(*********************************** G.D S.p.A. - Technical Department ***********************************
============= PROGRAM INFO ============
FOLDER:             TBD
MACHINES INVOLVED:  TBD 

============= DESCRIPTION =============
csp machine declaration

============= REVISIONS ===============
Date		Version	 	Author      	Description             
----------	-------		------------  	--------------------------------------------
2019/04/05 	0000.00	 	M.Grasso		Creation of the PRG

**********************************************************************************************************)
(*$R process_ref := prc; $*)
PROGRAM csp_case_transport_ls
VAR
	
	prc:											process;
	prc_path:										STRING;
	
END_VAR

_read_var_input();

_object_manager();

IF NOT objects_running()
THEN
	RETURN;	
END_IF

_read_process_image();

_mode_manager();

_set_runtime_properties();

(********************************* BODY *********************************)
(************************************************************************)

_handle_messages();

_write_output();

ACTION _handle_messages:
;
END_ACTION

ACTION _handle_process_test:
;
END_ACTION

ACTION _mode_manager:
IF process_mode_req_is_pending(prc)
THEN
    process_apply_mode_req_first_step(prc);
    CASE process_get_mode(prc) OF
        MODE_TO_ABSENT:
			;
        MODE_TO_INACTIVE:
			;
        MODE_TO_TEST:
			;
        MODE_TO_OPERATIONAL:
			;
    END_CASE
    process_apply_mode_req_second_step(prc);
END_IF
END_ACTION

ACTION _object_manager:
IF objects_initialization()
THEN
	sub_process_init(
		object_name					:= 'csp_case_transport_ls.prc', 
		process						:= csp_case_transport.prc, 
		CONVERSION_this				:= prc);
		
	prc_path 						:= process_get_path(prc);
END_IF

IF objects_running()
THEN
	process_cycle(prc);
END_IF
END_ACTION

ACTION _read_process_image:
;
END_ACTION

ACTION _read_var_input:
;
END_ACTION

ACTION _set_runtime_properties:
;
END_ACTION

ACTION _write_output:
;
END_ACTION

END_PROGRAM

(* stored: Version 1.1.0.1, ProductVersion 3.1.4022.12
   POU csp_case_transport_ls: Id {7285c901-0997-4019-8ca4-bf6088195d4a}, SpecialFunc None
   Action _handle_messages: Id {614d5296-bac9-4f40-9e45-5a318b044126}
   Action _handle_process_test: Id {2aaf7fe9-f453-4fc6-8b25-d63078fd3e93}
   Action _mode_manager: Id {c356dff1-5e85-4147-83e8-997d4070dfab}
   Action _object_manager: Id {dd527629-8a88-45e1-b784-1cdb905dd935}
   Action _read_process_image: Id {67b8af02-a294-4f7e-ac80-897a14e1a95f}
   Action _read_var_input: Id {7130963b-edf4-459a-8d3e-3eaa389ac302}
   Action _set_runtime_properties: Id {324673b3-7a09-4a01-8fd0-0a6aa14f2f55}
   Action _write_output: Id {b82c74ea-173f-4454-b3bf-89553765e2cc} *)
